(**************1个LED灯*************************)
FUNCTION_BLOCK FB_UVLed_R
VAR_INPUT
	single_double			:BOOL;//"Indicates unidirectional printing.TRUE IF the print is unidirectional, otherwise FALSE FOR bi-directional printing.
	initial_print_position	:INT;//"Indicates the initial print position: 0:from_home, 1:to_home."
	uv_power_leading		:DINT;//% "(leadingPower ConfigurePower-Settings method)Power to apply to leading LEDs of the UVUnit"
	uv_power_trailing		:DINT;//% "(trailingPower ConfigurePower-Settings method)Power to apply to trailing LEDs of the UVUnit"
	uvStart					:LREAL;//um "Position in micron where to start/stop curing depending on the direction (left/right)."	
	uvEnd					:LREAL;//mm "Position in micron where to start/stop curing depending on the direction (left/right)"
	ahead_pos				:LREAL:=100;//因YV灯有延迟，提前量uvEnd					:LREAL;//um "Position in micron where to start/stop curing depending on the direction (left/right)"	
	delay_pos				:LREAL:=100;//UV关闭延迟
	parts					:BYTE;
	
	Encoder					:LREAL;
	Moving					:BOOL;//fs MOVING
	FS_Direction_N			:BOOL;//反向
	FS_Direction_P			:BOOL;//正向
	//is_printing				:BOOL;
	UVError					:BOOL;
	IO_Error				:BOOL;
	UVisRemote				:BOOL;
END_VAR
VAR_OUTPUT
	state				:INT;
	error_code				:INT;
	uv_power		:DINT;//一个UV灯内 分段功率
	set_prats				:BYTE;//
	initialized			:BOOL;
	settings_applide		:BOOL;
	curing_started	:BOOL;
	curing_stopped	:BOOL;
	error					:BOOL;
	off					:BOOL;
	
END_VAR
VAR
	step				:INT;
	unidirection		:BOOL;//单向
	bidirectiona		:BOOL;//双向
	from_home			:BOOL;//Printing starts from the home position
	to_home				:BOOL;//Printing starts towards the home position
	error_trig1,error_trig2:Tc2_Standard.R_TRIG;
	uvStart_temp		:LREAL;
	uvEnd_temp			:LREAL;
	ton1:Tc2_Standard.TON;
END_VAR
VAR_IN_OUT
	Initialize				:BOOL;
	ConfigurePowerSettings	:BOOL;
	ConfigurePositions		:BOOL;
	StopCuring				:BOOL;
	SetOff					:BOOL;
END_VAR

set_prats:=parts;

(***************因YV灯有延迟，提前量****************************)
	uvStart_temp:=uvStart-ahead_pos;
	uvEnd_temp:=uvEnd+delay_pos;

CASE step OF
0://waiting
	IF Initialize THEN 
		step:=5;	
	ELSIF ConfigurePowerSettings THEN 
		step:=20;	
	ELSIF ConfigurePositions THEN 
		step:=40;
	ELSIF ConfigurePowerSettings THEN 
		step:=10;
	ELSIF StopCuring THEN 
		step:=40;
	ELSIF SetOff OR GVL.Reset THEN 
		step:=200;
	ELSIF state=UVLedStateEnum.ready_for_curing AND Moving THEN 
		step:=50;
	END_IF
	(******************状态自复位***************************)
	ton1(IN:=initialized OR  settings_applide OR  curing_started OR  curing_stopped 
				OR error OR  off , PT:=State_reset_time , Q=> , ET=> );
	IF ton1.Q THEN 
		initialized:=FALSE;
		settings_applide:=FALSE;
		curing_started:=FALSE;
		curing_stopped:=FALSE;
		error:=FALSE;
		off:=FALSE;
	END_IF
	
5://off
	state:=UVLedStateEnum.off;
	error_code:=UVLedErrorEnum.no_error;	
	uv_power:=0;
	
	ConfigurePowerSettings	:=FALSE;
	ConfigurePositions		:=FALSE;
	StopCuring				:=FALSE;
	SetOff					:=FALSE;
	bidirectiona			:=FALSE;
	from_home				:=FALSE;
	
	IF Initialize THEN 
		Initialize:=FALSE;
		state:=UVLedStateEnum.initializing;	
		step:=6;		
	END_IF
6://
	IF UVisRemote THEN 
		step:=10;	
	END_IF	
10://initializing	
	initialized:=TRUE;
	state:=UVLedStateEnum.ready;
	settings_applide:=FALSE;
	curing_started:=FALSE;
	curing_stopped:=FALSE;
	off:=FALSE;
	step:=0;
20://ready
	IF 	ConfigurePowerSettings THEN
		ConfigurePowerSettings:=FALSE; 
		IF single_double THEN 
			unidirection:=TRUE;
			bidirectiona:=FALSE;
		ELSE
			unidirection:=FALSE;
			bidirectiona:=TRUE;
		END_IF
		IF initial_print_position=1 THEN 
			to_home:=TRUE;
			from_home:=FALSE;
		ELSIF initial_print_position=0 THEN 
			to_home:=FALSE;
			from_home:=TRUE;
		END_IF
		state:=UVLedStateEnum.applying_settings;
		step:=30;
	END_IF
	IF SetOff OR GVL.Reset THEN	
		step :=200;
	END_IF
30://applying_settings
	ConfigurePowerSettings:=FALSE;	
	uv_power:=0;
	state:=UVLedStateEnum.settings_applied;
	settings_applide:=TRUE;
	step:=0;
40://settings_applied
	IF 	ConfigurePositions THEN 
		ConfigurePositions:=FALSE;
		IF uvStart>0 AND uvEnd>0   THEN 
			state:=UVLedStateEnum.ready_for_curing;
			step:=0;
		END_IF	
	END_IF
	IF StopCuring THEN 
		StopCuring:=FALSE;
		state:=UVLedStateEnum.ready;
		step:=0;
	END_IF
50://ready_for_curing
	//IF is_printing THEN 
		IF bidirectiona THEN 
			step:=60;
		ELSIF unidirection THEN 
			IF from_home THEN 
				step:=70;
			ELSIF to_home THEN 
				step:=80;
			END_IF
		END_IF
	//END_IF
60://bidirectiona   双向
	IF FS_Direction_P THEN 	//向右
		IF Encoder>=uvStart_temp  AND Encoder<=uvEnd_temp THEN    //右灯
			 uv_power:=uv_power_leading;
			 curing_started :=TRUE;
		ELSE uv_power:=0;
		END_IF	
		IF Encoder>uvEnd_temp  THEN  //结束
			curing_started :=FALSE;
			curing_stopped:=TRUE;
			step:=30;
		END_IF
	ELSIF FS_Direction_N THEN 
		IF Encoder>=uvStart_temp  AND Encoder<=uvEnd_temp THEN    //右灯
			 uv_power:=uv_power_trailing;
			 curing_started :=TRUE;
		ELSE uv_power:=0;
		END_IF
		IF Encoder<uvStart_temp  THEN  //结束
			curing_started :=FALSE;
			curing_stopped:=TRUE;
			step:=30;
		END_IF
	END_IF
	
	IF uv_power<>0 THEN 
		state:=UVLedStateEnum.curing;
	END_IF

	(*******范围内小车不运动*******)
	IF (Encoder>=uvStart_temp AND Encoder <=uvEnd_temp) AND NOT Moving (*OR NOT is_printing*)  THEN 
		uv_power:=0;
		curing_stopped:=TRUE;
		step:=30; 
	END_IF
70://unidirection/from_home
	IF FS_Direction_P THEN 
		IF Encoder>=uvStart_temp  AND Encoder<=uvEnd_temp THEN    //右灯
			 uv_power:=uv_power_leading;
			 curing_started :=TRUE;
		ELSE uv_power:=0;
		END_IF
		IF Encoder>uvEnd_temp  THEN  //结束
			curing_started :=FALSE;
			curing_stopped:=TRUE;
			step:=30;
		END_IF				
	END_IF
	
	IF uv_power<>0  THEN 
		state:=UVLedStateEnum.curing;
	END_IF
	IF FS_Direction_N THEN 
		uv_power:=0;
		curing_stopped:=TRUE;
		step:=30; 
	END_IF
	(*******范围内小车不运动*******)
	IF (Encoder>=uvStart_temp AND Encoder <=uvEnd_temp) AND NOT Moving (* OR NOT is_printing*)  THEN 
		uv_power:=0;
		curing_stopped:=TRUE;
		step:=30; 
	END_IF
	
80://unidirection/to_home
	IF FS_Direction_N THEN 
		IF Encoder>=uvStart_temp  AND Encoder<=uvEnd_temp THEN    //右灯
			 uv_power:=uv_power_trailing;
			 curing_started :=TRUE;
		ELSE uv_power:=0;
		END_IF
		IF Encoder<uvStart_temp  THEN  //结束
			curing_started :=FALSE;
			curing_stopped:=TRUE;
			step:=30;
		END_IF	
	END_IF
	
	IF uv_power<>0 THEN 
		state:=UVLedStateEnum.curing;
	END_IF
	IF FS_Direction_P THEN 
		uv_power:=0;
		curing_stopped:=TRUE;
		step:=30; 
	END_IF
	(*******范围内小车不运动*******)
	IF (Encoder>=uvStart_temp AND Encoder <=uvEnd_temp) AND NOT Moving  (*OR NOT is_printing*)  THEN 
		uv_power:=0;
		curing_stopped:=TRUE;
		step:=30; 
	END_IF
100://error
	state:=UVLedStateEnum.error;
	error:=TRUE;
	uv_power:=0;
	step:=0; 
	IF SetOff THEN	
		SetOff:=FALSE; 
		step :=200;
	END_IF
200://seting_off		
	SetOff:=FALSE; 
	state:=UVLedStateEnum.setting_off;
	error_code:=UVLedErrorEnum.no_error;
	uv_power:=0;
	off:=TRUE;
	state:=UVLedStateEnum.off;
	step:=0;
END_CASE
IF SetOff OR GVL.Reset THEN 
	step:=200;
END_IF

(*****************ERROR**************************************)
IF 	state<>UVLedStateEnum.setting_off AND state<>UVLedStateEnum.off AND state<>UVLedStateEnum.error THEN 
	error_trig1(CLK:=UVError AND state<>UVLedStateEnum.off , Q=> );
	error_trig2(CLK:=IO_Error AND state<>UVLedStateEnum.off , Q=> );
	IF GVL.Emstop_SAFE THEN 
		error_code:=UVLedErrorEnum.emergency_error;
		step:=100;
	ELSIF error_trig1.Q THEN 
		error_code:=UVLedErrorEnum.abnormal_temperature;
		step:=100;
	ELSIF error_trig2.Q THEN 
		error_code:=UVLedErrorEnum.unknown_error;
		step:=100;
	END_IF
END_IF

	(*******只要速度低于值，就不开灯*****)
IF ABS( Axis[FastScan].Ref.NcToPlc.ActVelo)<=10 THEN
	uv_power:=0;	
END_IF

END_FUNCTION_BLOCK

(* stored: Version 1.1.0.1, ProductVersion 3.1.4024.11
   POU FB_UVLed_R: Id {6da59c83-cf96-46ae-82df-ecf4a9801f30}, SpecialFunc None *)
